// ---- CNC Beckhoff/3 Control/HLI3_GetChannelActiveG.TcPOU
FUNCTION_BLOCK HLI3_GetChannelActiveG
VAR_INPUT
	bExec:	   BOOL;			// riding edge to start read
	nChanIdx: INT;    			// zero based channel index	
END_VAR
VAR_OUTPUT
	ActiveG : ARRAY[0..39] OF INT;
	bBusy: BOOL;
	bError: BOOL;
	nErrorID: UDINT;
END_VAR
VAR
	fbAdsRead: ADSREAD;
END_VAR

(* ========================================================= *)
(*    FUN: HLI3_GetChannelActiveG                   		 *)
(* --------------------------------------------------------- *)
(*   Desc: Gets the channel specific active G functions      *)
(*															 *)
(* Return: Array[0..39] filled with the G information (<> -1)*)
(* Author: MiB                                               *)
(*   Date: 12.01.2016                                        *)
(*   Rev.: 1.0                                               *)
(* ========================================================= *)

fbAdsRead(
	NETID:= '' , 
	PORT:= 553, 
	IDXGRP:= 16#20100 + INT_TO_UDINT(nChanIdx) + 1, 
	IDXOFFS:= 16#3C , 
	LEN:= SIZEOF(ActiveG) , 
	DESTADDR:= ADR(ActiveG),
	READ:= bExec, 
	TMOUT:= , 
	BUSY=> bBusy, 
	ERR=> bError, 
	ERRID=> nErrorId );

END_FUNCTION_BLOCK

// ---- CNC Beckhoff/3 Control/HLI3_GetChannelMessage.TcPOU
FUNCTION_BLOCK HLI3_GetChannelMessage
VAR_INPUT
	/// Number of channel 
	nChanIdx: INT;
	bExecute: BOOL := FALSE;
	bShowDlg: BOOL := FALSE;
END_VAR
VAR_OUTPUT
	strToPLC: STRING(HLI_MSG_CONTENT_STRL) := '';
	iMsgType: DWORD := 0;
END_VAR
VAR
	pChannel: POINTER TO HIGH_LEVEL_INTERFACE_CH;
	pMsgCU: POINTER TO MC_CONTROL_MSG_UNIT;
	pMsgToPLC: POINTER TO STRING(HLI_MSG_CONTENT_STRL);
END_VAR

(* ========================================================= *)
(*     FB: HLI_GetChannelMessage                             *)
(* --------------------------------------------------------- *)
(*   Desc: Get message from the CNC                          *)
(*   Author: MK, MiB                                         *)
(*   Date: 20.11.2012                                        *)
(*   Last:                                                   *)
(*   Rev.: 1.01                                              *)
(* ========================================================= *)

IF NOT HLI3_CheckChannelValid(nChannel := nChanIdx) THEN
	RETURN;
END_IF


(* Get pointer to data of a specific channel at the HLI *)
pChannel := gpCh[nChanIdx];

(* Control unit at the HLI that handles channel specific messages *)
pMsgCU := ADR(pChannel^.msg_mc_control);

IF bExecute = TRUE THEN
	(* Is the complete message in the control unit? *)
	IF pMsgCU^.request_semaphor_rw = TRUE
	THEN
		(* Pointer to content of the message sent to the PLC *)
		pMsgToPLC := ADR(pMsgCU^.request_r.inhalt);

		(* Get the message from the control unit *)
		strToPLC := pMsgToPLC^;

   	    CNCSystem.Channel[nChanIdx].Message := strToPLC;

		(* Get the message type *)
		iMsgType := pMsgCU^.request_r.typ;

		(* Pop up dialog with the message send to the PLC *)
		IF bShowDlg THEN
			ADSLOGSTR( msgCtrlMask := ADSLOG_MSGTYPE_MSGBOX OR ADSLOG_MSGTYPE_LOG,
			           msgFmtStr   := 'Message sent to PLC via HLI:%s',
			           strArg      := strToPLC);
		END_IF

		(* Acknowledge that you got the message *)
		pChannel^.msg_mc_control.request_semaphor_rw  := FALSE;
	END_IF;
END_IF;

END_FUNCTION_BLOCK

// ---- CNC Beckhoff/3 Control/HLI3_GetEtherCATAxisInfo.TcPOU
FUNCTION HLI3_GetEtherCATAxisInfo : ST_DriveRef
VAR
	arrTemp: ARRAY[1..24] OF BYTE;
	arrNetIdAchse2: ARRAY[0..MAX_STRING_LENGTH] OF BYTE;
	i: INT;
	id: DINT;
	nCha: UINT;
	nPort: UINT;
END_VAR
VAR_INPUT
	nHliAxisIdx: INT;
END_VAR

(* ========================================================= *)
(*    FUN: HLI_GetEtherCATAxisInfo                   		 *)
(* --------------------------------------------------------- *)
(*   Desc: Gets the information about a SoE Drive (Ax5000)   *)
(*  benötigt: TcEtherCAT.lib   *)
(* Return: Structure with the information for the drive     *)
(* Author: MiB                                               *)
(*   Date: 20.11.2012                                        *)
(*   Rev.: 1.2                                               *)
(* ========================================================= *)


IF NOT HLI3_CheckAxisValid(nHliAxisIdx := nHliAxisIdx) THEN
	HLI3_GetEtherCATAxisInfo.sNetId := '';
	HLI3_GetEtherCATAxisInfo.nDriveNo := 0;
	HLI3_GetEtherCATAxisInfo.nSlaveAddr := 0;
	RETURN;	
END_IF


HLI3_GetEtherCATAxisInfo.sNetId := gpAx[nHliAxisIdx]^.lr_state.twincat_box.ads_netid_r;
HLI3_GetEtherCATAxisInfo.nDriveNo := UINT_TO_BYTE(gpAx[nHliAxisIdx]^.lr_state.twincat_box.channel_r);
HLI3_GetEtherCATAxisInfo.nSlaveAddr :=gpAx[nHliAxisIdx]^.lr_state.twincat_box.ads_port_r;

RETURN;

END_FUNCTION

// ---- CNC Beckhoff/3 Control/HLI3_GetFeedholdState.TcPOU
FUNCTION HLI3_GetFeedholdState : BOOL
VAR_INPUT
	/// Number of channel 
	nChanIdx: INT;
END_VAR


IF NOT HLI3_CheckChannelValid(nChannel := nChanIdx) THEN
	RETURN;
END_IF
HLI3_GetFeedholdState:=gpCh[nChanIdx]^.bahn_mc_control.feedhold.state_r;

END_FUNCTION

// ---- CNC Beckhoff/3 Control/HLI3_GetIpoState.TcPOU
FUNCTION HLI3_GetIpoState : BOOL
VAR_INPUT
	nChanIdx: INT;
END_VAR



IF NOT HLI3_CheckChannelValid(nChannel := nChanIdx) THEN
	RETURN;
END_IF

HLI3_GetIpoState:=gpCh[nChanIdx]^.bahn_state.interpolation_active_r;

END_FUNCTION

// ---- CNC Beckhoff/3 Control/HLI3_SetAxisGantryOn.TcPOU
FUNCTION HLI3_SetAxisGantryOn : BOOL
VAR_INPUT
	nHliAxisIdx: INT;
	bEnable: BOOL;
END_VAR

(****************************************************************************************)
(* POU:		HLI_SetAxisGantryOn                      									*)
(* Type:	Function																	*)
(* Author: 	HR																			*)
(* Date: 	11/01/24																	*)
(* Rev.: 	1.0																			*)
(* ------------------------------------------------------------------------------------ *)
(* Desc:	Enables the axis specific control unit for driving out the gantry			*)
(*			difference. The actual movement is triggered by the input 'bEnable'.		*)
(*			The current axis has to be a gantry slave. That means:						*)
(*				+ It is not attached to a channel										*)
(*				+ kenngr.achs_mode		0x2000n		(where n specifies the axis type)	*)
(*				+ kenngr.gantry_ax_nr	1			(e. g. axis no. of gantry master)	*)
(*				+ kenngr.gantry_offset  10000		(e. g. difference to be driven out)	*)
(*				+ kenngr.gantry_vb_korr	20000		(e. g. velocity for driving out)	*)
(****************************************************************************************)

(* Check specified logical axis no first *)
IF NOT HLI3_CheckAxisValid(nHliAxisIdx := nHliAxisIdx) THEN
	HLI3_SetAxisGantryOn := FALSE;
	RETURN;
END_IF

gpAx[nHliAxisIdx]^.lr_mc_control.gantry_on.enable_w	:= TRUE;
gpAx[nHliAxisIdx]^.lr_mc_control.gantry_on.command_w	:= bEnable;
HLI3_SetAxisGantryOn	:= TRUE;

END_FUNCTION

// ---- CNC Beckhoff/3 Control/HLI3_SetAxisReferenceCam.TcPOU
FUNCTION HLI3_SetAxisReferenceCam : BOOL
VAR_INPUT
	nHliAxisIdx: INT;
	bReferenceCam: BOOL;
END_VAR
VAR
	/// Index of axis specific HLI area 
	nHliAxIfcIdx: INT;
END_VAR

(* ========================================================= *)
(*    FUN: HLI_SetAxisReferenceCam                           *)
(* --------------------------------------------------------- *)
(*   Desc:                                                   *)
(* Author: MK,MiB                                            *)
(*   Date: 30.11.2012                                        *)
(*   Rev.: 1.1                                               *)
(* ========================================================= *)


IF NOT HLI3_CheckAxisValid(nHliAxisIdx := nHliAxisIdx) THEN
	HLI3_SetAxisReferenceCam := FALSE;
	RETURN;
END_IF

(* set reference cam *)
gpAx[nHliAxisIdx]^.lr_mc_control.reference_cam.enable_w  := TRUE;
gpAx[nHliAxisIdx]^.lr_mc_control.reference_cam.command_w := bReferenceCam;

HLI3_SetAxisReferenceCam := TRUE;

END_FUNCTION

// ---- CNC Beckhoff/3 Control/HLI3_SetAxisReferencePosition.TcPOU
FUNCTION HLI3_SetAxisReferencePosition : BOOL
VAR_INPUT
	bSetRefpos: BOOL;
	nHliAxisIdx: INT;
END_VAR

(* ========================================================= *)
(*    FUN: HLI_SetAxisReferenceposition                      *)
(* --------------------------------------------------------- *)
(*   Desc:                                                   *)
(* Author: HR                                                *)
(*   Date: 09.11.2010                                        *)
(*   Rev.: 1.0                                               *)
(* ========================================================= *)
HLI3_SetAxisReferencePosition := FALSE;

IF NOT HLI3_CheckAxisValid(nHliAxisIdx := nHliAxisIdx) THEN	
	RETURN;
END_IF

(* set reference position *)
gpAx[nHliAxisIdx]^.lr_mc_control.set_reference_position.command_w := bSetRefpos;
HLI3_SetAxisReferencePosition := TRUE;

END_FUNCTION

// ---- CNC Beckhoff/3 Control/HLI3_SetAxisSpindleStopAtProgramEnd.TcPOU
FUNCTION_BLOCK HLI3_SetAxisSpindleStopAtProgramEnd
VAR_INPUT
	bExecute: BOOL;
	bSpindelStopAtProgramEnd: BOOL;
	nHliAxisIdx: INT;
END_VAR
VAR_OUTPUT
	bBusy: BOOL;
END_VAR
VAR
	/// Index of axis specific HLI area 
	nHliAxIfcIdx: INT;
	nState: INT;
	fbRTrigExecute: R_TRIG;
END_VAR

(****************************************************************************************)
(* POU:		HLI_SetAxisSpindleStopAtProgramEnd                      					*)
(* Type:		FB																		*)
(* Author: 	HR                                              							*)
(* Date: 	24.01.11																	*)
(* Rev.: 	1.0                                               							*)
(* ------------------------------------------------------------------------------------ *)
(* Desc:	Check wether the axis specified by input 'nLogAxisNo' is a spindle and 		*)
(*			(re-) sets (depending on the state of input 'bSpindelStopAtProgramEnd') 	*)
(*			the spindle stop feature on the HLI.										*)
(****************************************************************************************)

(****************************************************************************************)
(*								Check logical axis no									*)
(****************************************************************************************)
IF NOT HLI3_CheckAxisValid(nHliAxisIdx := nHliAxisIdx) THEN	
	RETURN;
END_IF
(****************************************************************************************)
(*									Build trigger										*)
(****************************************************************************************)
fbRTrigExecute
	(CLK := bExecute);

(****************************************************************************************)
(*								   (Re-)set sequence									*)
(****************************************************************************************)
CASE nState OF
 (* ----------------------------------------------------------------------------------- *)
 0: (* INIT STATE  *)
  	bBusy			:= FALSE;

	IF fbRTrigExecute.Q THEN
		bBusy		:= TRUE;
		nState		:= 10;
	END_IF

 (* ----------------------------------------------------------------------------------- *)
 10: (* ENABLE THE CONTROL UNIT IF THE AXIS IS A SPINDLE *)

	IF gpAx[nHliAxisIdx]^.ipo_state.spindle_axis_r THEN
		gpAx[nHliAxisIdx]^.ipo_mc_control.spdl_stop_at_prog_end.enable_w := TRUE;
		nState 		:= 20;
	ELSE
		nState 		:= 0;
	END_IF

 (* ---------------------------------------------------------------------------------- *)
 20: (* (RE-) SET SPINDLE STOP FUNCTION *)
	gpAx[nHliAxisIdx]^.ipo_mc_control.spdl_stop_at_prog_end.command_w := bSpindelStopAtProgramEnd;
	nState 			:= 0;
END_CASE

END_FUNCTION_BLOCK

// ---- CNC Beckhoff/3 Control/HLI3_SetAxisTrackingOperation.TcPOU
FUNCTION HLI3_SetAxisTrackingOperation : BOOL
VAR_INPUT
	nHliAxisIdx: INT;
	bPLCAxisEnable: BOOL;
END_VAR

(* ========================================================= *)
(*    FUN: HLI_SetAxisTrackingOperation                      *)
(* --------------------------------------------------------- *)
(*   Desc:                                                   *)
(*   Author: TV                                              *)
(*   Date: 15.09.2006                                        *)
(*   Rev.: 1.0                                               *)
(*         1.1 13.08.2013 Nachführbetrieb nicht bei Achsfehler einschalten *)
(* ========================================================= *)

IF NOT HLI3_CheckAxisValid(nHliAxisIdx := nHliAxisIdx) THEN	
	HLI3_SetAxisTrackingOperation := FALSE;
	RETURN;
END_IF

(* tracking operation (follow up) on / off *)
IF NOT bPLCAxisEnable THEN
	gpAx[nHliAxisIdx]^.lr_mc_control.follow_up.command_w := TRUE;
		HLI3_SetAxisTrackingOperation := TRUE;
ELSE
	gpAx[nHliAxisIdx]^.lr_mc_control.follow_up.command_w := FALSE;
		HLI3_SetAxisTrackingOperation := FALSE;
END_IF

END_FUNCTION

// ---- CNC Beckhoff/3 Control/HLI3_SetProbingSignal.TcPOU
FUNCTION HLI3_SetProbingSignal : BOOL
VAR_INPUT
	nHliAxisIdx: INT;
	bProbingSignal: BOOL;
END_VAR


IF NOT HLI3_CheckAxisValid(nHliAxisIdx := nHliAxisIdx) THEN	
	HLI3_SetProbingSignal := FALSE;
	RETURN;
END_IF


gpAx[nHliAxisIdx]^.lr_mc_control.probing_signal.enable_w  := TRUE;
gpAx[nHliAxisIdx]^.lr_mc_control.probing_signal.command_w := bProbingSignal;
HLI3_SetProbingSignal := TRUE;

END_FUNCTION

// ---- CNC Beckhoff/4 MHT-Function/HLI3_QuitAxisMFunction.TcPOU
FUNCTION HLI3_QuitAxisMFunction : BOOL
VAR_INPUT
	/// Number of axis 
	nHliAxisIdx: INT;
END_VAR
VAR
	/// Data of a M/H techno unit 
	pMHProcess: POINTER TO HLI_M_H_PROZESS;
	/// Data of a spindle unit 
	pSProcess: POINTER TO HLI_S_PROZESS;
	/// Data of a techno unit 
	pTProcess: POINTER TO HLI_T_PROZESS;
	/// local pointer to Data of actual Axis 
	pAxisData: POINTER TO HIGH_LEVEL_INTERFACE_AX;
	/// local pointer to actual techno unit 
	pActTechnoUnit: POINTER TO TECHNO_UNIT_AX;
	/// loop variable 
	idx: UINT;
	/// Index of axis specific technology function at HLI 
	nTechFctMaxIdx: UINT;
	/// basis id of a tool 
	nToolBasicId: UDINT;
	/// spindle movement command 
	SpdlMoveCmd: UINT;
	/// SpindleRevolution 
	Revolution: UDINT;
	/// SpindleRevolution 
	pRevolution: POINTER TO UDINT;
	/// Number of M-function 
	FuncNr: UDINT;
END_VAR

(* ========================================================= *)
(*    FUN: HLI_QuitAxisMFunction                             *)
(* --------------------------------------------------------- *)
(*   Desc:                                                   *)
(* Author: MK                                                *)
(*   Rev.: 1.1                                               *)
(*   Date: 18.07.2002                                        *)
(*       : 08.04.2005                                        *)
(* ========================================================= *)

HLI3_QuitAxisMFunction := FALSE;
IF NOT (HLI3_CheckAxisValid(nHliAxisIdx := nHliAxisIdx)) THEN
	RETURN;
END_IF


(* get pointer to Axis data *)
pAxisData := gpAx[nHliAxisIdx];

(* test if there are open synchronisations  *)
IF pAxisData^.used_units_std_sync_r > 0 THEN

	nTechFctMaxIdx := pAxisData^.used_units_std_sync_r - 1;

	FOR idx := 0 TO nTechFctMaxIdx DO
	
		(* get pointer to actual techno unit *)
		pActTechnoUnit := ADR(pAxisData^.techno_unit_std_sync[idx]);
	
		(* test if this M-function has to be acknowledged *)
		IF pActTechnoUnit^.please_rw = TRUE AND				(* request from CNC *)
			pActTechnoUnit^.done_w = FALSE					(* not acknowledged *)
		THEN
	
			IF pActTechnoUnit^.fkt_ctrl_r = HLI_INTF_M_FKT THEN
				(* Example: read number of M-function *)
				pMHProcess := ADR(pActTechnoUnit^.attribut_r.data[0]);
				FuncNr := pMHProcess^.nr;
				ADSLOG(strMsg:='Axis acknowledge of M-function: %d', nDINT:=UDINT_TO_DINT(FuncNr), strArg:='');
			ELSE
				IF pActTechnoUnit^.fkt_ctrl_r = HLI_INTF_SPINDEL THEN (* spindle-fuction *)
					pSProcess := ADR(pActTechnoUnit^.attribut_r.data[0]);
	
					(* Example: read revolution of S-function *)
					Revolution := DINT_TO_UINT(pSProcess^.rev);
					ADSLOG(strMsg:='Spindle S-function: %d', nDINT:=UDINT_TO_DINT(Revolution), strArg:='');
	
					(* Example: read number of S-function *)
					SpdlMoveCmd := pSProcess^.move_cmd;
					ADSLOG(strMsg:='Spindle acknowledge of M-function: %d', nDINT:=SpdlMoveCmd, strArg:='');
				ELSE
					ADSLOGDINT( msgCtrlMask :=    ADSLOG_MSGTYPE_MSGBOX
					                           OR ADSLOG_MSGTYPE_LOG,
								msgFmtStr   := 'Axis acknowledge unknown type: %d',
								dintArg     := pActTechnoUnit^.fkt_ctrl_r);
				END_IF
			END_IF
	
			(* acknowledge this M-function *)
			pActTechnoUnit^.please_rw := FALSE;
			pActTechnoUnit^.done_w := TRUE;
	
			HLI3_QuitAxisMFunction := TRUE;
		END_IF
	END_FOR

END_IF

END_FUNCTION

// ---- CNC Beckhoff/4 MHT-Function/PRG_FastMFunctions.TcPOU
PROGRAM PRG_FastMFunctions
VAR
	anMFunctionNo						: ARRAY[0..MAX_FAST_M_FUNC_ITEM_IDX] OF UINT;
	
	fbFastMFunctionProvider				: HLI3_FastMFunctionProvider;
	fbFastMFunctionHandler				: HLI3_FastMFunctionHandler;
	
	(* abyOutput					AT %Q*	: ARRAY[0..MAX_FAST_M_FUNC_OUTPUT_IDX] OF BYTE; *) 
	abyOutput					: ARRAY[0..MAX_FAST_M_FUNC_OUTPUT_IDX] OF BYTE; (* Demo output, if needed use the line above *)

END_VAR

(****************************************************************************************)
(* POU:		PRG_FastMFunctions                    										*)
(* Type:	PRG																			*)
(* Author: 	RCH		                                             						*)
(* Date: 	14/10/29																	*)
(* Rev.: 	1.0                                               							*)
(* ------------------------------------------------------------------------------------ *)
(* Desc.:	PLC program to demonstrate usage of MOS_TS M functions using the FB´s		*)
(*			HLI3_FastMFunctionProvider and HLI3_FastMFunctionHandler.					*)
(*			In order to achieve a determenistic output behavior this program has to be 	*)
(*			called by a task running synchronously to the CNC GEO task. Therefore that	*)
(*			task´s priority  has to be adjusted in a way that it gets called by the 	*)
(* 			realtime system	right after the CNC GEO task.								*)
(*																						*)
(*			THIS IMPLEMENTATION REQUIRES A 1MS CNC GEO AND 1MS FAST PLC TASK CYCLE!!!	*)
(* ------------------------------------------------------------------------------------ *)
(* Rev.:	<Enter revision number here>												*)
(* Date:	<Enter revision data here>				                                   	*)
(* Author:	<Enter author´s shortcut here>											 	*)
(* Desc.:	<Enter description here>													*)
(****************************************************************************************)


(****************************************************************************************)
(*	  						Configure M function no´s to provide						*)
(****************************************************************************************)
(* Add up to MAX_FAST_M_FUNC_ITEM_IDX m function numbers that should be handled by 		*)
(* fbFastMFunctionProvider.																*)
anMFunctionNo[0]	:= 25;
anMFunctionNo[1]	:= 26;

fbFastMFunctionProvider
	(nHliChanIdx	:= 0, 
	 anMFunctionNo	:= anMFunctionNo
	);
	
(****************************************************************************************)
(*	  						 	Handle Laser ON/OFF (M25/M26)							*)
(****************************************************************************************)
(* M function numbers for switching ON and OFF have to be contained in the 				*)
(* 'anMFunctionNo' array of the HLI3_FastMFunctionProvider instance which provides the	*)
(* 'stData' structure to this FB.														*)
(* The delay times nDelayOn and nDelayOff can be used to adopt to external hardware		*)
(* delays!																				*)
fbFastMFunctionHandler
	(bForceOff		:= FALSE, 
	 bReset			:= FALSE, 
	 nFunctionNoOn	:= 25, 
	 nDelayOn		:= 0,			
	 nFunctionNoOff	:= 26, 
	 nDelayOff		:= 0,
	 stData			:= fbFastMFunctionProvider.stData,
	 abyOutput		=> abyOutput
	);

END_PROGRAM

// ---- CNC Beckhoff/5 Variables/HLI3_GetVEChannelDIntValue.TcPOU
FUNCTION HLI3_GetVEChannelDIntValue : DINT
VAR_INPUT
	/// HLI Channel Index 
	nChanIdx: INT;
	/// Index of variable  range 1 ...     HLI_VE_VALUEMAX 
	nVEIndex: DINT;
	/// Array index. 0 if no array 
	nArrayIndex: DINT := 0;
	/// serves acess to the global variable array 
	bGlobal: BOOL;
END_VAR
VAR
	pVeData: POINTER TO VEData := 0;
	/// Size of the datatype of the returned value 
	iDatatypeSize: DINT;
	ptr: POINTER TO DINT;
	ChIdx: UDINT;
	SizeField: DINT := 0;
END_VAR

(* ========================================================= *)
(*    FUN: GetVEChannelDINTValue                            *)
(* --------------------------------------------------------- *)
(*   Desc: Reads a V.E.Variable of DINT                    *)
(* 	 Author: CL  / TV                                        *)
(*   Date: 16.05.2006                                        *)
(*   Last: 28.01.2013                                        *)
(*   Rev.: 1.3                                               *)
(* ========================================================= *)

IF  nVEIndex >= 0 AND
	nArrayIndex >= 0 THEN

	(* test if channel specific or global *)
	IF bGlobal = FALSE  THEN
		IF NOT HLI3_CheckChannelValid(nChannel := nChanIdx) THEN
			RETURN;
		END_IF
				
		pVeData := gpVECh[nChanIdx];
	ELSE
		pVeData := gpVEGlobal;
	END_IF

	IF pVeData <> 0 THEN
		IF pVeData <> 0 THEN
			iDatatypeSize := SIZEOF(ptr^);
                         	ptr := pVeData +  24  * nVEIndex + (iDatatypeSize * nArrayIndex);
                           HLI3_GetVEChannelDIntValue := ptr^; (* successfully completed return *)
                END_IF
	END_IF
END_IF

END_FUNCTION

// ---- CNC Beckhoff/5 Variables/HLI3_GetVEChannelBooleanValue.TcPOU
FUNCTION HLI3_GetVEChannelBooleanValue : BOOL
VAR_INPUT
	/// HLI Channel Index
	nChanIdx: INT;
	/// Index of variable  range 1 ...     HLI_VE_VALUEMAX 
	nVEIndex: DINT;
	/// Array index. 0 if no array 
	nArrayIndex: DINT := 0;
	/// serves acess to the global variable array 
	bGlobal: BOOL;
END_VAR
VAR
	pVeData: POINTER TO VEData := 0;
	/// Size of the datatype of the returned value 
	iDatatypeSize: DINT;
	ptr: POINTER TO BOOL;
	ChIdx: UDINT;
	SizeField: DINT := 0;
END_VAR

(* ========================================================= *)
(*    FUN: GetVEChannelDINTValue                            *)
(* --------------------------------------------------------- *)
(*   Desc: Reads a V.E.Variable of Boolean                   *)
(* 	 Author: CL  / TV                                        *)
(*   Date: 16.05.2006                                        *)
(*   Last: 05.12.2013                                        *)
(*   Rev.: 1.3                                               *)
(* ========================================================= *)

IF  nVEIndex >= 0 AND
	nArrayIndex >= 0 THEN

	(* test if channel specific or global *)
	IF bGlobal = FALSE  THEN
		IF NOT HLI3_CheckChannelValid(nChannel := nChanIdx) THEN
			RETURN;
		END_IF
				
		pVeData := gpVECh[nChanIdx];
	ELSE
		pVeData := gpVEGlobal;
	END_IF

	IF pVeData <> 0 THEN
		IF pVeData <> 0 THEN
			iDatatypeSize := SIZEOF(ptr^);
                         	ptr := pVeData +  24  * nVEIndex + (iDatatypeSize * nArrayIndex);
                           HLI3_GetVEChannelBooleanValue := ptr^; (* successfully completed return *)
                END_IF
	END_IF
END_IF

END_FUNCTION

// ---- CNC Beckhoff/5 Variables/HLI3_GetVEChannelLRealValue.TcPOU
FUNCTION HLI3_GetVEChannelLRealValue : LREAL
VAR_INPUT
	/// HLI Channel Index
	nChanIdx: INT;
	/// Index of variable  range 1 ...     HLI_VE_VALUEMAX 
	nVEIndex: DINT;
	/// Array index. 0 if no array 
	nArrayIndex: DINT := 0;
	/// serves acess to the global variable array 
	bGlobal: BOOL;
END_VAR
VAR
	pVeData: POINTER TO VEData := 0;
	/// Size of the datatype of the returned value 
	iDatatypeSize: DINT;
	ptr: POINTER TO LREAL;
	ChIdx: UDINT;
	SizeField: DINT := 0;
END_VAR

(* ========================================================= *)
(*    FUN: GetVEChannelLrealValue                            *)
(* --------------------------------------------------------- *)
(*   Desc: Reads a V.E.Variable of REAL64                    *)
(* 	 Author: CL  / TV                                        *)
(*   Date: 16.05.2006                                        *)
(*   Last: 28.01.2013                                        *)
(*   Rev.: 1.3                                               *)
(* ========================================================= *)

IF  nVEIndex >= 0 AND
	nArrayIndex >= 0 THEN

	(* test if channel specific or global *)
	IF bGlobal = FALSE  THEN
		IF NOT HLI3_CheckChannelValid(nChannel := nChanIdx) THEN
			RETURN;
		END_IF
				
		pVeData := gpVECh[nChanIdx];
	ELSE
		pVeData := gpVEGlobal;
	END_IF

	IF pVeData <> 0 THEN
		IF pVeData <> 0 THEN
			iDatatypeSize := SIZEOF(ptr^);
                         	ptr := pVeData +  24  * nVEIndex + (iDatatypeSize * nArrayIndex);
                           HLI3_GetVEChannelLRealValue := ptr^; (* successfully completed return *)
                END_IF
	END_IF
END_IF

END_FUNCTION

// ---- CNC Beckhoff/5 Variables/HLI3_GetVEChannelStringValue.TcPOU
FUNCTION HLI3_GetVEChannelStringValue : STRING(23)
VAR_INPUT
	/// HLI Channel Index
	nChanIdx: INT;
	/// Index of variable  range 1 ...     HLI_VE_VALUEMAX 
	nVEIndex: DINT;
	/// Array index. 0 if no array 
	nArrayIndex: DINT := 0;
	/// serves acess to the global variable array 
	bGlobal: BOOL;
END_VAR
VAR
	pVeData: POINTER TO VEData := 0;
	/// Size of the datatype of the returned value 
	iDatatypeSize: DINT;
	ptr: POINTER TO STRING(24);
	ChIdx: INT;
END_VAR

(* ========================================================= *)
(*    FUN: GetVEChannelStringValue                           *)
(* --------------------------------------------------------- *)
(*   Desc: Reads a V.E.Variable of STRING                    *)
(* 	 Author: CL / TV                                         *)
(*   Date: 16.05.2006                                        *)
(*   Last: 28.01.013                                        *)
(*   Rev.: 1.1                                               *)
(* ========================================================= *)

(* Config Example
	VAR[0].name                                           StringValue
	VAR[0].index                                           1
	VAR[0].TYPE                                           STRING
	VAR[0].scope                                          GLOBAL
	VAR[0].synchronisation                                TRUE
	VAR[0].access_rights                                  READ_WRITE
	VAR[0].array_size                                     21
	VAR[0].size                                           24
	VAR[0].create_hmi_interface                           0
*)

IF  nVEIndex >= 0 AND
	nArrayIndex >= 0 THEN

	(* test if channel specific or global *)
	IF bGlobal = FALSE  THEN
		IF NOT HLI3_CheckChannelValid(nChannel := nChanIdx) THEN
			RETURN;
		END_IF
		pVeData := gpVECh[nChanIdx];
	ELSE
		pVeData := gpVEGlobal;
	END_IF

	IF pVeData <> 0 THEN
		 IF pVeData <> 0 THEN
			iDatatypeSize := SIZEOF(ptr^);
			iDatatypeSize := 24;
            ptr := pVeData +  24  * nVEIndex + (iDatatypeSize * nArrayIndex);
            HLI3_GetVEChannelStringValue := ptr^; (* successfully completed return *)
         END_IF
	END_IF
END_IF

END_FUNCTION

// ---- CNC Beckhoff/5 Variables/HLI3_LinkVEChannelStructure.TcPOU
FUNCTION HLI3_LinkVEChannelStructure : POINTER TO DWORD
VAR_INPUT
	/// HLI Channel Index 
	nChanIdx: INT;	
	/// serves acess to the global variable array 
	bGlobal: BOOL;
END_VAR
VAR
	pVeData: POINTER TO VEData := 0;
	ptr: POINTER TO DWORD;
	ChIdx: UDINT;
	nVEIndex: POINTER TO DWORD;
END_VAR

(* ========================================================= *)
(*    FUN: LinkVEChannelStructure                            *)
(* --------------------------------------------------------- *)
(*   Desc: Link VE variable to the memory of the CNC         *)
(*   Author: CL, MK                                            *)
(*   Date: 16.05.2006                                        *)
(*   Rev.: 1.3                                               *)
(*       : MK  access changed                                *)
(*		   1.2												 *)
(*		   MiB 7.11.2012 check zero pointers				 *)
(*		   TV 19.08.2015 Input Parm. nIndex removed          *) 
(* ========================================================= *)

	(* test if channel specific or global *)
     IF bGlobal THEN
    	IF gpVEGlobal = 0  THEN   (* check for  zero pointer *)
        	RETURN; (* Cancel *)
        END_IF
			pVeData := gpVEGlobal;
	 ELSE
		IF NOT HLI3_CheckChannelValid(nChannel := nChanIdx) THEN
			RETURN;
		END_IF
							
		pVeData := gpVECh[nChanIdx];
	END_IF 

	IF pVeData <> 0 THEN
    	ptr := pVeData;
		HLI3_LinkVEChannelStructure := ptr; (* successfully completed return *)
	END_IF

END_FUNCTION

// ---- CNC Beckhoff/5 Variables/HLI3_SetVEChannelDIntValue.TcPOU
FUNCTION HLI3_SetVEChannelDIntValue : BOOL
VAR_INPUT
	/// HLI Channel Index
	nChanIdx: INT;
	/// Index of variable  range 1 ...     HLI_VE_VALUEMAX 
	nVEIndex: DINT;
	/// Array index. 0 if no array 
	nArrayIndex: DINT := 0;
	/// serves acess to the global variable array 
	bGlobal: BOOL;
	/// Value to be written 
	val: DINT;
END_VAR
VAR
	pVeData: POINTER TO VEData := 0;
	/// Size of the datatype of the returned value 
	iDatatypeSize: DINT;
	ptr: POINTER TO DINT;
	ChIdx: UDINT;
	SizeField: DINT := 0;
END_VAR

(* ========================================================= *)
(*    FUN: SetVEChannelDIntValue                           *)
(* --------------------------------------------------------- *)
(*   Desc: Writes a V.E.Variable of REAL64                    *)
(* 	 Author: CL  / TV                                        *)
(*   Date: 16.05.2006                                        *)
(*   Last: 28.01.2013                                        *)
(*   Rev.: 1.3                                               *)
(* ========================================================= *)

IF  nVEIndex >= 0 AND
	nArrayIndex >= 0 THEN

	(* test if channel specific or global *)
	IF bGlobal = FALSE  THEN
		IF NOT HLI3_CheckChannelValid(nChannel := nChanIdx) THEN
			RETURN;
		END_IF
				
		pVeData := gpVECh[nChanIdx];
	ELSE
		pVeData := gpVEGlobal;
	END_IF

	IF pVeData <> 0 THEN
		IF pVeData <> 0 THEN
			iDatatypeSize := SIZEOF(ptr^);
            ptr := pVeData +  24  * nVEIndex + (iDatatypeSize * nArrayIndex);
			ptr^:=val;
            HLI3_SetVEChannelDIntValue := TRUE; (* successfully completed return *)						  						   
       	END_IF
	END_IF
END_IF

END_FUNCTION

// ---- CNC Beckhoff/5 Variables/HLI3_SetVEChannelBooleanValue.TcPOU
FUNCTION HLI3_SetVEChannelBooleanValue : BOOL
VAR_INPUT
	/// HLI Channel Index
	nChanIdx: INT;
	/// Index of variable  range 1 ...     HLI_VE_VALUEMAX 
	nVEIndex: DINT;
	/// Array index. 0 if no array 
	nArrayIndex: DINT := 0;
	/// serves acess to the global variable array 
	bGlobal: BOOL;
	/// Value to be written 
	val: BOOL;
END_VAR
VAR
	pVeData: POINTER TO VEData := 0;
	/// Size of the datatype of the returned value 
	iDatatypeSize: DINT;
	ptr: POINTER TO BOOL;
	ChIdx: UDINT;
	SizeField: DINT := 0;
END_VAR

(* ========================================================= *)
(*    FUN: SetVEChannelDIntValue                           *)
(* --------------------------------------------------------- *)
(*   Desc: Writes a V.E.Variable of REAL64                    *)
(* 	 Author: CL  / TV                                        *)
(*   Date: 16.05.2006                                        *)
(*   Last: 05.12.2013                                        *)
(*   Rev.: 1.3                                               *)
(* ========================================================= *)

IF  nVEIndex >= 0 AND
	nArrayIndex >= 0 THEN

	(* test if channel specific or global *)
	IF bGlobal = FALSE  THEN
		IF NOT HLI3_CheckChannelValid(nChannel := nChanIdx) THEN
			RETURN;
		END_IF
				
		pVeData := gpVECh[nChanIdx];
	ELSE
		pVeData := gpVEGlobal;
	END_IF

	IF pVeData <> 0 THEN
		IF pVeData <> 0 THEN
			iDatatypeSize := SIZEOF(ptr^);
            ptr := pVeData +  24  * nVEIndex + (iDatatypeSize * nArrayIndex);
			ptr^:=val;
            HLI3_SetVEChannelBOOLeanValue := TRUE; (* successfully completed return *)						  						   
       	END_IF
	END_IF
END_IF

END_FUNCTION

// ---- CNC Beckhoff/5 Variables/HLI3_SetVEChannelLRealValue.TcPOU
FUNCTION HLI3_SetVEChannelLRealValue : BOOL
VAR_INPUT
	/// HLI Channel Index
	nChanIdx: INT;
	/// Index of variable  range 1 ...     HLI_VE_VALUEMAX 
	nVEIndex: DINT;
	/// Array index. 0 if no array 
	nArrayIndex: DINT := 0;
	/// serves acess to the global variable array 
	bGlobal: BOOL;
	/// Value to be written 
	val: LREAL;
END_VAR
VAR
	pVeData: POINTER TO VEData := 0;
	/// Size of the datatype of the returned value 
	iDatatypeSize: DINT;
	ptr: POINTER TO LREAL;
	ChIdx: UDINT;
	SizeField: DINT := 0;
END_VAR

(* ========================================================= *)
(*    FUN: SetVEChannelLrealValue                           *)
(* --------------------------------------------------------- *)
(*   Desc: Writes a V.E.Variable of REAL64                    *)
(* 	 Author: CL  / TV                                        *)
(*   Date: 16.05.2006                                        *)
(*   Last: 06.03.2012                                        *)
(*   Rev.: 1.3                                               *)
(* ========================================================= *)

IF  nVEIndex >= 0 AND
	nArrayIndex >= 0 THEN

	(* test if channel specific or global *)
	IF bGlobal = FALSE  THEN
		IF NOT HLI3_CheckChannelValid(nChannel := nChanIdx) THEN
			RETURN;
		END_IF
				
		pVeData := gpVECh[nChanIdx];
	ELSE
		pVeData := gpVEGlobal;
	END_IF

	IF pVeData <> 0 THEN
		IF pVeData <> 0 THEN
			iDatatypeSize := SIZEOF(ptr^);
            ptr := pVeData +  24  * nVEIndex + (iDatatypeSize * nArrayIndex);
			ptr^:=val;
            HLI3_SetVEChannelLRealValue := TRUE; (* successfully completed return *)						  						   
       	END_IF
	END_IF
END_IF

END_FUNCTION

// ---- CNC Beckhoff/5 Variables/HLI3_SetVEChannelStringValue.TcPOU
FUNCTION HLI3_SetVEChannelStringValue : BOOL
VAR_INPUT
	/// HLI Channel Index
	nChanIdx: INT;
	/// Index of variable  range 1 ...     HLI_VE_VALUEMAX 
	nVEIndex: DINT;
	/// Array index. 0 if no array 
	nArrayIndex: DINT := 0;
	/// Value to be written 
	val: STRING(23);
	/// serves acess to the global variable array 
	bGlobal: BOOL;
END_VAR
VAR
	pVeData: POINTER TO VEData := 0;
	/// Size of the datatype of the returned value 
	iDatatypeSize: DINT;
	ptr: POINTER TO STRING;
	ChIdx: INT;
END_VAR

(* ========================================================= *)
(*    FUN: SetVEChannelStringValue                           *)
(* --------------------------------------------------------- *)
(*   Desc: Writes a V.E.Variable of STRING                   *)
(* 	 Author: CL / TV                                         *)
(*   Date: 16.05.2006                                        *)
(*   Last : 13.12.2012										 *)
(*   Rev.: 1.1                                               *)
(* ========================================================= *)

(* Config Example
	VAR[0].name                                           StringValue
	VAR[0].index                                           1
	VAR[0].TYPE                                           STRING
	VAR[0].scope                                          GLOBAL
	VAR[0].synchronisation                                TRUE
	VAR[0].access_rights                                  READ_WRITE
	VAR[0].array_size                                     21
	VAR[0].size                                           24
	VAR[0].create_hmi_interface                           0
*)

IF  nVEIndex >= 0 AND
	nArrayIndex >= 0 THEN

	(* test if channel specific or global *)
	IF bGlobal = FALSE  THEN
		IF NOT HLI3_CheckChannelValid(nChannel := nChanIdx) THEN
			RETURN;
		END_IF
				
		pVeData := gpVECh[nChanIdx];
	ELSE
		pVeData := gpVEGlobal;
	END_IF

	IF pVeData <> 0 THEN
		iDatatypeSize := SIZEOF(ptr^);
		iDatatypeSize := 24;
        ptr := ADR(pVeData^)  +  24  * nVEIndex + (iDatatypeSize * (nArrayIndex));
        ptr^ := val; (* successfully completed return *)
		HLI3_SetVEChannelStringValue := TRUE;
	END_IF
END_IF

END_FUNCTION

// ---- CNC Beckhoff/9 Mis/FB_WriteCNCZeroOffset.TcPOU
/// ------------------------------------------------------------------------------------ 
/// Desc:	Description																	
///**************************************************************************************
///**************************************************************************************
///	 Write NPV Value directly to CNC core using V.G. Variables via ADS	
///**************************************************************************************
FUNCTION_BLOCK FB_WriteCNCZeroOffset
VAR_INPUT
	/// rising edge to start 
	bExecute: BOOL;
	/// which table, G54=1, G55=2, G55=3, .... 
	nG159Index: BYTE;
	/// Channel Indedx
	nChanIdx: UDINT;
	/// Axis name in channel 
	sAxisName: STRING(95);
	/// value to set 
	lrValue: LREAL;
END_VAR
VAR_OUTPUT
	bBusy: BOOL;
	bError: BOOL;
	nErrorID: UDINT;
END_VAR
VAR
	fbAdsWrite: ADSWRITE;
	stCNCG159VG: ST_CNCG159VG;
END_VAR

stCNCG159VG.dValue := LREAL_TO_DINT(lrValue * 10000);
stCNCG159VG.sTarget := 'V.G.NP[';
stCNCG159VG.sTarget := CONCAT(stCNCG159VG.sTarget, BYTE_TO_STRING(nG159Index));
stCNCG159VG.sTarget := CONCAT(stCNCG159VG.sTarget, '].V.');
stCNCG159VG.sTarget := CONCAT(stCNCG159VG.sTarget,sAxisName);

fbAdsWrite(
	PORT:= 552 ,
	IDXGRP:= 16#22300 + nChanIdx+1,
	IDXOFFS:=16#3F,
	LEN:= SIZEOF(stCNCG159VG) ,
	SRCADDR:=ADR(stCNCG159VG) ,
	WRITE:= bExecute,
	TMOUT:= ,
	BUSY=> bBusy,
	ERR=> bError ,
	ERRID=> nErrorID);

END_FUNCTION_BLOCK

// ---- CNC Beckhoff/9 Mis/FB_WriteCNCZeroOffsetDefault.TcPOU
/// ------------------------------------------------------------------------------------ 
/// Desc:	Description																	
///**************************************************************************************
///**************************************************************************************
///	 Write NPV Default (the active table afetr reset) directly to CNC core using V.G. Variables via ADS	
///**************************************************************************************
FUNCTION_BLOCK FB_WriteCNCZeroOffsetDefault
VAR_INPUT
	/// rising edge to start 
	bExecute: BOOL;
	/// which table, G54=1, G55=2, G55=3, .... 
	nG159Index: BYTE;
	/// Channel Indedx
	nChanIdx: UDINT;
END_VAR
VAR_OUTPUT
	bBusy: BOOL;
	bError: BOOL;
	nErrorID: UDINT;
END_VAR
VAR
	fbAdsWrite: ADSWRITE;
	stCNCG159VG: ST_CNCG159VG;
END_VAR

stCNCG159VG.dValue := nG159Index;
stCNCG159VG.sTarget := 'V.G.NP_DEFAULT';

fbAdsWrite(
	PORT:= 552 ,
	IDXGRP:= 16#22300 + nChanIdx+1,
	IDXOFFS:=16#3F,
	LEN:= SIZEOF(stCNCG159VG) ,
	SRCADDR:=ADR(stCNCG159VG) ,
	WRITE:= bExecute,
	TMOUT:= ,
	BUSY=> bBusy,
	ERR=> bError ,
	ERRID=> nErrorID);

END_FUNCTION_BLOCK

// ---- CNC Beckhoff/9 Mis/HLI3_CheckCNCAlive.TcPOU
PROGRAM HLI3_CheckCNCAlive
VAR_INPUT
	nChanIdx: INT;
END_VAR

VAR
	bMessageDisplayed : BOOL;
END_VAR

(* The assumption is made that the cycle time of the PLC is at least twice as big as the CNC cycle time.

The Cycle time of CNC is displayed in element:
	pMC[1]^.addr^.HLIHeadChannel_Data.LCWatchDogUnit_lc.D_cycle_time_r

remark: Take care if PLC cycle is smaller not to check CNC faster as possible !!!

To simulate failure of CNC set cycle time of PLC smaller than CNC (Resource/task configuration).
*)

// HLI3_CheckCNCAlive := FALSE;
IF NOT HLI3_CheckChannelValid(nChannel := nChanIdx) THEN
	RETURN;
END_IF
 
(* Copy current state of live sign to watchdog state    *)
gpCh[nChanIdx]^.head.lc_watchdog.alive_rw
	:= gpCh[nChanIdx]^.head.lc_watchdog.alive_rw;

IF gpCh[nChanIdx]^.head.lc_watchdog.alive_rw = FALSE AND NOT bMessageDisplayed THEN
	(* PLC detects CNC not alive -> start individual emergency stop within PLC *)
	ADSLOGSTR( msgCtrlMask := ADSLOG_MSGTYPE_ERROR OR
							ADSLOG_MSGTYPE_MSGBOX OR
							ADSLOG_MSGTYPE_LOG,
			msgFmtStr := 'PLC detects CNC not alive: %s',
			strArg := 'channel 1');
			
			bMessageDisplayed := TRUE;
END_IF


(* assign return value *)
//HLI3_CheckCNCAlive := gpCh[nChanIdx]^.head.lc_watchdog.alive_rw;

(* reset live sign for next cycle *)
gpCh[nChanIdx]^.head.lc_watchdog.alive_rw := FALSE;

END_PROGRAM

// ---- CNC Beckhoff/9 Mis/HLI3_GetLogAxisId.TcPOU
FUNCTION HLI3_GetLogAxisId : INT
VAR_INPUT
	nHliAxisIdx: INT;
END_VAR
VAR
	i: INT;
END_VAR

(* ========================================================= *)
(*    FUN: HLI3_GetLogAxisId                            	 *)
(* --------------------------------------------------------- *)
(*   Desc: returns the Log. Axis Idx for a given HLI Index   *)
(*   Author: TV                                              *)
(*   Date: 22.01.2014                                        *)
(*   Rev.: 1.0                                               *)
(* ========================================================= *)
HLI3_GetLogAxisId := -1;
IF NOT HLI3_CheckAxisValid(nHliAxisIdx := nHliAxisIdx) THEN
	RETURN;
END_IF

HLI3_GetLogAxisId := UINT_TO_INT(gpAx[nHliAxisIdx]^.head.log_ax_nr_r);

END_FUNCTION

// ---- CNC Beckhoff/9 Mis/HLI_HandleMessages.TcPOU
FUNCTION_BLOCK HLI_HandleMessages
VAR_INPUT
	/// Enable 
	bEnable: BOOL;
	/// Number of channel 
	nChanIdx: INT;
	/// Channelstruct 
	pChannel: POINTER TO ST_CncChannel;
END_VAR
VAR_OUTPUT
	bNewMessage: BOOL;
	bError: BOOL;
	sMessage: STRING(255);
END_VAR
VAR
	/// Index of channel specific HLI area 

	bFirstCycle: BOOL := TRUE;
	bModeChanged: BOOL;
	nState: USINT;
	nActMode: UDINT;
	dwCncState: DWORD;
	fbRtrigStateStart: R_TRIG;
	pString: POINTER TO STRING(HLI_MSG_CONTENT_STRL);
	fbLog: ADSLOGEVENT;
	stMessageData: TcEvent;
END_VAR
VAR CONSTANT
	sFormat: STRING(2) := '%s';
END_VAR

(******************************************************************************)
(* Name:		HLI_HandleMessages											 	*)
(* Date:		08/12/01													 	*)
(* Author:	H. Rausch (Beckhoff Automation GmbH)							 	*)
(* Ver:		1.0																	*)
(* Desc:		Function block for recieving messages from CNC and passing them to*)
(*				the TwinCAT EventLogger. Only the latest message from CNC is 	*)
(*				active there. The event will be resetted if a new message from	*)
(*				CNC is recieved, the CNC state changes to 'ACTIVE', the CNC mode*)
(*				is changed or the channel is resetted							*)
(*																				*)
(*				Messages are passed as a fill string to the event logger with 	*)
(*				source id 9000 and event id 1. This requires a correspondant 	*)
(*				configuration in the tceventsourcelocation.xml and in an		*)
(*				associated message file!										*)
(* ---------------------------------------------------------------------------*)
(* Rev:		Add new version number here!										*)
(* Date.		Add revision data here											*)
(* Desc:		Add revision description here!									*)
(******************************************************************************)

(* Write event config data once on start up *)
IF bFirstCycle THEN
	stMessageData.bQuitRequired			:= TRUE;
	stMessageData.Class					:= TCEVENTCLASS_MESSAGE;
	stMessageData.DataFormatStrAddress	:= ADR(sFormat);
	stMessageData.Prio					:= 0;
	stMessageData.Id					:= 1;
	stMessageData.SourceId 				:= 9000;
	stMessageData.Flags 				:= TCEVENTFLAG_LOG OR TCEVENTFLAG_SRCID;
	stMessageData.StreamType			:= TCEVENTSTREAM_SIMPLE;
	stMessageData.ProgId 				:= 'TcEventFormatter.TcXmlFormatter';
END_IF



(* Check for zero pointer and leave fb if necessary *)
IF NOT HLI3_CheckChannelValid(nChannel := nChanIdx) THEN
	RETURN;
END_IF
	(* Check CNC state *)
	dwCncState := HLI3_GetChannelState(nChanIdx:=nChanIdx);

	(* Rising trig if CNC state changes to ACTIVE *)
	fbRtrigStateStart
		(CLK := (dwCncState = HLI_IMCM_PROCESS_ACTIVE));

	(* Watch CNC mode *)
	bModeChanged	:= (nActMode <> pChannel^.ActMode);
	nActMode 		:= pChannel^.ActMode;

IF NOT bEnable THEN
	gpCh[nChanIdx]^.msg_mc_control.enable_w				:= FALSE;
	gpCh[nChanIdx]^.msg_mc_control.request_semaphor_rw	:= FALSE;
	sMessage										:= '';
ELSE
	gpCh[nChanIdx]^.msg_mc_control.enable_w 			:= TRUE;

	CASE nState OF
	 0:
		(* Wait for new messages from CNC *)
		IF gpCh[nChanIdx]^.msg_mc_control.request_semaphor_rw THEN
			(* Convert byte stream to string *)
			pString  := ADR(gpCh[nChanIdx]^.msg_mc_control.request_r.inhalt);
			sMessage := pString^;
			(* Reset notification from HLI *)
			gpCh[nChanIdx]^.msg_mc_control.request_semaphor_rw := FALSE;

			nState := 1;
		END_IF

	 1:
		(* Wait that ADSEVENTLOG instance is cleared *)
		IF (fbLog.EventState = 0) THEN
			nState := 2;
		END_IF

	 2:
		(* Set message to eventlogger *)
		IF (fbLog.EventState > 0) THEN
			nState := 0;
		END_IF

	END_CASE

	(* Managing Eventlogger *)
	fbLog
		(NETID				:= '',
		 PORT					:= 110,
		 Event				:= (nState = 2),
		 EventQuit			:= (nState = 1) OR
									(dwCncState = HLI_IMCM_PROCESS_RESETTING) OR
									fbRtrigStateStart.Q OR
									bModeChanged,
		 EventConfigData	:= stMessageData,
		 EventDataAddress	:= ADR(sMessage),
		 EventDataLength	:= SIZEOF(sMessage),
		 TMOUT				:= t#2s
		);
END_IF

(* Reset first cycle indicator *)
bFirstCycle := FALSE;

END_FUNCTION_BLOCK

// ---- CNC Beckhoff/9 Mis/HLI_MoveSpindle.TcPOU
///*********************************************************************************************************
///NAME.......................:	HLI_MoveSpindle	
///DATUM....................:	7.9.2009
///AUTOR....................:	Michael Balsfulland (MiB)
///VERSION................:	1.0
///				1.1 20.8.2010 MiB: kompletter Umbau auf Schrittkette mit Fehlerhandling
///BESCHREIBUNG.:	 Spindel mit einer vorgegeben Geschwindigkeit starten oder Spindel stoppen
///......................: 	
///
///**********************************************************************************************************
FUNCTION_BLOCK HLI_MoveSpindle
VAR
	pUnit: POINTER TO MC_CONTROL_EXT_TO_IPO;
	fbRTrigStart: R_TRIG;
	fbRTrigStop: R_TRIG;
	nState: INT;
	/// Index of axis specific HLI area 
	nHliAxIfcIdx: UDINT;
END_VAR
VAR_INPUT
	/// Spindel Achssnummer 
	nLogAxisNr: UDINT;
	/// U/min 
	nSpeed: DINT;
	/// steigende Flanke 
	bStart: BOOL;
	/// steigende Flanke 
	bStop: BOOL;
END_VAR
VAR_OUTPUT
	bBusy: BOOL;
	bError: BOOL;
	nErrID: INT;
	sErrText: STRING;
END_VAR

fbRTrigStart(clk := bStart);
IF fbRTrigStart.Q THEN
	bError := FALSE;
	nErrId := 0;
	sErrText := '';
	nState := 100;   (* Spindel starten *)
END_IF


fbRTrigStop(clk := bStop);
IF fbRTrigStop.Q THEN
	bError := FALSE;
	nErrId := 0;
	sErrText := '';
	nState := 200;  (* Spindel stoppen *)
END_IF

nHliAxIfcIdx := nLogAxisNr - 1;

IF fbRTrigStop.Q OR fbRTrigStart.Q THEN   (* Grundzustände testen *)
	bBusy := TRUE;
	IF nLogAxisNr = 0 THEN
		nState := -1;
		nErrID := 1;
		sErrText := 'Spindel ID = 0';
	END_IF
	IF ADR(gpAx[nHliAxIfcIdx]^)  = 0  THEN
		nState := -1;
		nErrID := 2;
		sErrText := 'Achsstruktur nicht vorhanden -> eventuell HLI Init nicht OK';
	END_IF
	IF gpAx[nHliAxIfcIdx]^.ipo_state.spindle_axis_r <> TRUE THEN
		nState := -1;
		nErrID := 3;
		sErrText := 'Achse ist kene Spindel';
	END_IF
END_IF

CASE nState OF


-1: (* Fehler *)
   	bError := TRUE;
	bBusy := FALSE;

0: (* IDLE *)
	bBusy := FALSE;


100: (* Spindel starten *)
	(* Check Override *)
	gpAx[nHliAxIfcIdx]^.ipo_mc_control.override.enable_w := TRUE;
	IF gpAx[nHliAxIfcIdx]^.ipo_mc_control.override.state_r = 0 THEN
		nState := -1;
		nErrID := 4;
		sErrText := 'Spindeloverride = 0';
	ELSE
		nState := 110;
	END_IF


110: (* Parametrieren des Aufrufs *)
	pUnit := ADR(gpAx[nHliAxIfcIdx]^.ipo_mc_control.ext_to_ipo);
	IF (nSpeed > 0) THEN
		pUnit^.command_w.vb_prog   :=  nSpeed * 360 / 60 * 1000  ;(*Programmierter Satzvorschub in u/min*)
		pUnit^.command_w.dreh_info := 1;(* rechtslauf *)
	ELSE
		pUnit^.command_w.vb_prog   :=  nSpeed * 360 / 60 * 1000  ;(*Programmierter Satzvorschub in u/min*)
		pUnit^.command_w.dreh_info := 0;(* linkslauf*)
	END_IF
	pUnit^.command_w.geo_gm_fkt    := 0;(*G- und M- Fkt.-Bitleiste*)
	pUnit^.command_w.satz_typ      := HLI_NC_MOVE_ENDLOS;(*Einer der Werte: HLI_NC_MOVE_LIN, HLI_NC_MOVREF, HLI_NC_MOVE_ENDLOS, HLI_NC_SPINDEL_STOP*)
	IF pUnit^.command_semaphor_rw = FALSE THEN
	    pUnit^.command_semaphor_rw := TRUE;
	    nState := 120;
	END_IF

	IF (nSpeed=0) THEN
		nState := -1;
		nErrID := 6;
		sErrText := 'Vorgabegeschwindigkeit = 0';
	END_IF

120: (* Start *)

	IF pUnit^.command_semaphor_rw = FALSE THEN
	    nState := 300;  (* checken Auftragsfehler *)
	END_IF



200: (* Spindel Stopp*)
	pUnit := ADR(gpAx[nHliAxIfcIdx]^.ipo_mc_control.ext_to_ipo);
	pUnit^.command_w.satz_typ  := HLI_NC_SPINDEL_STOP;(*Einer der Werte: HLI_NC_MOVE_LIN, HLI_NC_MOVREF, HLI_NC_MOVE_ENDLOS, HLI_NC_SPINDEL_STOP*)
	pUnit^.command_w.dreh_info := 0;(*Drehinformation*)
	IF pUnit^.command_semaphor_rw = FALSE THEN
	    pUnit^.command_semaphor_rw := TRUE;
	    nState := 210;
	END_IF

210: (* Warten auf Stop *)
	IF pUnit^.command_semaphor_rw = FALSE THEN
	    nState := 300;   (* checken Auftragsfehler *)
	END_IF

300: (* checken Auftragsfehler *)
	IF (gpAx[nHliAxIfcIdx]^.ipo_state.spindle_order_error_r) THEN
		nState := -1;
		nErrID := 5;
		sErrText := 'Beauftragunsfehler Spindel';
	ELSE
		nState := 310;
	END_IF

310: (* Warten auf Solldrehzahl erreicht *)

	IF (gpAx[nHliAxIfcIdx]^.lr_state.rev_erreicht_r) THEN
		nState := 0;
	END_IF


END_CASE


(*
IF nLogAxisNr <> 0 THEN
	IF pAC[nLogAxisNr] <> 0  THEN
		IF ADR(gpAx[nLogAxisNr]^) <> 0  THEN
			IF gpAx[nLogAxisNr]^.ipo_state.X_SpindleAxis = TRUE THEN

				(* command spindle revolution *)
				IF fbRTrigStart.Q THEN
					pCommand := ADR(gpAx[nLogAxisNr]^.ipo_mc_control.MCControlExtToIpo_ExtToIpo);
					IF (nSpeed > 0) THEN
						pCommand^.command_w.D_VbProg :=  DINT_TO_UDINT((nSpeed * 360 / 60) * 1000)  ;(*Programmierter Satzvorschub in u/min*)
  						pCommand^.command_w.W_DrehInfo := 1;(* rechtslauf *)
					ELSE
						pCommand^.command_w.D_VbProg :=  DINT_TO_UDINT((-nSpeed * 360 / 60) * 1000)  ;(*Programmierter Satzvorschub in u/min*)
						pCommand^.command_w.W_DrehInfo := 0;(* linkslauf*)
					END_IF
					pCommand^.command_w.D_GeoGmFkt := 0;(*G- und M- Fkt.-Bitleiste*)
					pCommand^.command_w.W_SatzTyp := HLI_NC_MOVE_ENDLOS;(*Einer der Werte: HLI_NC_MOVE_LIN, HLI_NC_MOVREF, HLI_NC_MOVE_ENDLOS, HLI_NC_SPINDEL_STOP*)
					pCommand^.command_semaphor_rw := TRUE;
				END_IF
				(* command spindle revolution *)
				IF fbRTrigStop.Q THEN
					pCommand := ADR(gpAx[nLogAxisNr]^.ipo_mc_control.MCControlExtToIpo_ExtToIpo);
					pCommand^.command_w.D_VbProg := 600000000;(*Programmierter Satzvorschub*)
					pCommand^.command_w.D_GeoGmFkt := 0;(*G- und M- Fkt.-Bitleiste*)

					pCommand^.command_w.W_SatzTyp := HLI_NC_SPINDEL_STOP;(*Einer der Werte: HLI_NC_MOVE_LIN, HLI_NC_MOVREF, HLI_NC_MOVE_ENDLOS, HLI_NC_SPINDEL_STOP*)
					pCommand^.command_w.W_DrehInfo := 0;(*Drehinformation*)
					pCommand^.command_semaphor_rw := TRUE;
				END_IF
			END_IF
		END_IF
	END_IF
END_IF
*)

END_FUNCTION_BLOCK

// ---- CNC Beckhoff/9 Mis/PB_10_CNC_Spindelkopplung.TcPOU
PROGRAM PB_10_CNC_Spindelkopplung
VAR
	pCoupling: POINTER TO HLI_COMMAND_AXIS_COUPLING;
	p_AxisCouplingState: POINTER TO HLI_STATE_AXIS_COUPLING;
	nState: INT;
	bBusy: BOOL;
	fbRTrig: R_TRIG;
	bCouple: BOOL;
	fbFTrig: F_TRIG;
END_VAR

(* allow axis coupling *)
gpAx[5]^.lr_mc_control.axis_coupling.enable_w := TRUE;


pCoupling := ADR(gpAx[5]^.lr_mc_control.axis_coupling.command_w);
p_AxisCouplingState := ADR(gpAx[5]^.lr_mc_control.axis_coupling.state_r);


fbRTrig(clk := bCouple);
fbFTrig(clk := bCouple);


IF (fbRTrig.Q) THEN			(* start coupling *)
	pCoupling^.desc[0].mode  := HLI_AXIS_COUPLING_DIRECT;
	pCoupling^.desc[0].ax_nr := 5;
	bBusy := TRUE;
	nState := 10;
END_IF


IF (fbFTrig.Q) THEN		(* end coupling *)
	pCoupling^.desc[0].mode  := HLI_AXIS_COUPLING_INACTIVE;
	pCoupling^.desc[0].ax_nr := 0;
	bBusy := TRUE;
	nState := 10; 
END_IF




CASE nState OF

0: (*IDLE *)
	bBusy := FALSE;


10: (* Koppeln oder Enkoppeln starten *)
	pCoupling^.semaphor_rw := TRUE;
	nState := nState + 10;

20:	(* Warten auf Koppeln fertig *)
	IF (pCoupling^.semaphor_rw = FALSE) THEN
		nState := 0;
	END_IF


END_CASE

END_PROGRAM

// ---- CNC Beckhoff/9 Mis/HLI3_ResetSpindle.TcPOU
FUNCTION HLI3_ResetSpindle : BOOL
VAR_INPUT
	/// axis number of spindle 
	nHliAxisIdx: INT;
END_VAR
VAR
	/// Index of axis specific HLI area 
	nHliAxIfcIdx: INT;
	SpdlState: BOOL;
	SpdlCommand: BOOL;
	ResetCmd: BOOL := FALSE;
	/// local pointer to data of actual axis 
	pResetUnit: POINTER TO MC_CONTROL_BOOL_UNIT;
END_VAR

HLI3_ResetSpindle := FALSE;

IF NOT HLI3_CheckAxisValid(nHliAxisIdx := nHliAxisIdx) THEN
	HLI3_ResetSpindle := FALSE;
	RETURN;
END_IF

	pResetUnit := ADR(gpAx[nHliAxisIdx]^.ipo_mc_control.spdl_reset);
	SpdlState  := pResetUnit^.state_r;

	IF ResetCmd = TRUE THEN
		pResetUnit^.command_w := TRUE;
		SpdlCommand           := pResetUnit^.command_w;
		HLI3_ResetSpindle          := SpdlState;
	END_IF

END_FUNCTION

// ---- CNC Beckhoff/Demo/PRG_Demo.TcPOU
PROGRAM PRG_Demo
VAR
	sLine1: STRING;
	sLine2: STRING;
	fbWriteZeroFddefault: FB_WriteCNCZeroOffsetDefault;
	bTest: BOOL;
	fbReadActiceG: HLI3_GetChannelActiveG;
	
	bReadG: BOOL;
	
END_VAR

PRG_MachineStatusV2();


sLine1 := 'Test line 1';
sLine2 := 'Test line two';

fbWriteZeroFddefault(
	bExecute:= bTest, 
	nG159Index:= 5 , 
	nChanIdx:=0, 
	bBusy=> , 
	bError=> , 
	nErrorID=> );
	
	
fbReadActiceG(
	bExec:= bReadG, 
	nChanIdx:= 0 , 
	ActiveG=> , 
	bBusy=> , 
	bError=> , 
	nErrorID=> );	
	
;

END_PROGRAM

// ---- CNC Beckhoff/Demo/PRG_MachineStatusV2.TcPOU
PROGRAM PRG_MachineStatusV2
VAR	
	fbTon: TON;
	fbTon2: TON;
	btest: BOOL;
	sName: STRING;
	sFarbe: STRING;
	nFarbe : UDINT;
	nFarbe2: UDINT;
	value: UDINT;
	value2 : UDINT;
	bUp: BOOL;
END_VAR


fbTon(in := NOT fbton.Q, pt := t#250ms);
IF (fbTon.Q) THEN
	btest := NOT bTest;
END_IF

fbton2(in := NOT fbton2.Q, pt := t#30ms);
IF fbton2.Q THEN

	IF (bUp) THEN
		value := value + 1;
	ELSE
		value := value - 1;
	END_IF
	IF value >= 200 THEN
		bUp := FALSE;
		value := 200;
	END_IF
	IF value <= 0 THEN
		bUp := TRUE;
		value := 0;
	END_IF
	value2 := 100 - value;
END_IF

nFarbe2 := 16#FF000000 + value2 * 2 * 16#010000 + value * 2 * 16#01;

IF btest THEN
	sName := 'EIN';
	sFarbe := 'blau';
	nFarbe := 16#FF0000FF;
ELSE
	sName := 'aus';
	sFarbe := 'rot';
	nFarbe := 16#FFFF0000;

END_IF

END_PROGRAM

// ---- CNC Beckhoff/Messages/FB_EventLog.TcPOU
FUNCTION_BLOCK FB_EventLog
VAR_INPUT
	bEvent: BOOL;
	bEventQuit: BOOL;
	bReset: BOOL;
	eLogMethod: E_LogMethod := Static;
	nSourceId: UDINT;
	nEventId: UDINT;
	nEventDataAddr: UDINT;
	nEventDataSize: UDINT;
	sFormat: STRING;
END_VAR
VAR_OUTPUT
	nEventState: UDINT;
	bEventActive: BOOL;
	bError: BOOL;
	nErrorId: UDINT;
END_VAR
VAR
	bEventInternal: BOOL;
	bEventActiveInternal: BOOL;
	fbFtrigEvent: F_TRIG;
	fbRtrigEvent: R_TRIG;
	fbRtrigEventInternal: R_TRIG;
	stEventData: TcEvent;
	fbEventLogger: ADSLOGEVENT;
END_VAR

(******************************************************************************)
(* 								 Konfiguration des Events									*)
(******************************************************************************)
stEventData.Flags 					:= TCEVENTFLAG_LOG OR TCEVENTFLAG_SRCID OR TCEVENTFLAG_FMTSELF OR 16#1000;
stEventData.StreamType				:= TCEVENTSTREAM_SIMPLE;
stEventData.ProgId 					:= 'TcEventFormatter.TcXmlFormatter';
stEventData.Id 						:= nEventId;
stEventData.SourceId 				:= nSourceId;
stEventData.DataFormatStrAddress	:= ADR(sFormat);
stEventData.bQuitRequired 			:= TRUE;

(******************************************************************************)
(* 					Interne Bildung des eventausloesenden Signals					*)
(******************************************************************************)
fbFtrigEvent
	(CLK := bEvent);

fbRtrigEvent
	(CLK := bEvent);

bEventInternal	:= (bEvent AND (eLogMethod = Static)) OR
					   (fbFtrigEvent.Q AND (eLogMethod = FallingTrig)) OR
					   (fbRtrigEvent.Q AND (eLogMethod = RisingTrig));

fbRtrigEventInternal
	(CLK := bEventInternal);

IF fbRtrigEventInternal.Q THEN
	bEventActiveInternal	:= TRUE;
ELSIF (fbEventLogger.EventState > 0) THEN
	bEventActiveInternal	:= FALSE;
END_IF

(******************************************************************************)
(* 							  Uebergabe an den Eventlogger								*)
(******************************************************************************)
fbEventLogger
	(NETID						:= '',
	 PORT						:= 110,
	 Event						:= bEventInternal,
	 EventQuit					:= bEventQuit,
	 EventConfigData			:= stEventData,
	 EventDataAddress			:= nEventDataAddr,
	 EventDataLength			:= nEventDataSize,
	 FbCleanup 					:= bReset,
	 TMOUT						:= t#2s,
	 EventState					=> nEventState,
	 Err						=> bError,
	 ErrId						=> nErrorId
	);

bEventActive					:= (fbEventLogger.EventState > 0) OR bEventActiveInternal;

END_FUNCTION_BLOCK

// ---- CNC Beckhoff/Messages/FB_ExtSimpleEventLog.TcPOU
///****************************************************************************************
///Name:				FB_ExtSimpleEventLog
///Date:				13.10.2004
///Author:			Dirk Nordberg (BECKHOFF INDUSTRIE ELEKTRONIK)
///
///Description: Function block to control the EventLogger
///	Messages can be activated or deactivated through an array of bool.
///	The subscription of the array is equivalent to EventID from EventLogger.
///	Funtion block will be initialized with Init flag, then the busy flag is set true. 
///
///	Revision:	1.3
///	History:		13.10.2004	Ng	start coding
///				17.04.2005	MK	runtime optimized
///				06.09.2005 	MiB extended version (renamed to FB_ExtSimpleEventLog)

///****************************************************************************************
FUNCTION_BLOCK FB_ExtSimpleEventLog
VAR_INPUT
	/// Rising flag starts the initialization 
	Init: BOOL;
	/// Alarm error class 
	Class: UINT;
	/// Activate or deaktivate confirmation 
	QuitRequired: BOOL;
	/// Adress of the array for the messages 
	adrAlarmArray: POINTER TO BOOL;
	/// ...with constant boundaries ARRAY_LBOUND to ARRAY_UBOUND for array size 
	adrQuitArray: POINTER TO BOOL;
	/// ...with constant boundaries ARRAY_LBOUND to ARRAY_UBOUND for array size 
	adrEventData: POINTER TO ST_EventData;
END_VAR
VAR_OUTPUT
	Busy: BOOL;
	Err: BOOL;
	ErrId: UDINT;
END_VAR
VAR CONSTANT
	ARRAY_LBOUND: UDINT := FIRST_MESSAGE;
	ARRAY_UBOUND: UDINT := LAST_MESSAGE;
	TCEVENTDATAFORMATSTRING: STRING(80) := ' ';
	STATE_INIT: INT := 0;
	STATE_IDLE: INT := 1;
	STATE_RESET_EVENT: INT := 2;
	STATE_QUIT_EVENT: INT := 3;
	STATE_RESET_END: INT := 4;
	STATE_WAIT: INT := 5;
END_VAR
VAR
	state: INT;
	///{flag nowatch on }
	bReady: BOOL;
	nMsgHasChanged: DINT;
	bEvtState: ARRAY[ARRAY_LBOUND..ARRAY_UBOUND] OF BOOL;
	event: ARRAY[ARRAY_LBOUND..ARRAY_UBOUND] OF ADSLOGEVENT;
	idx: UDINT;
	CfgEvent: TcEvent;
	bWait: BOOL;
	ptAlarm: POINTER TO BOOL;
	ptQuit: POINTER TO BOOL;
	RT_Init: R_TRIG;
	ptData: POINTER TO ST_EventData;
	stDummy: ST_EventData;
	/// Format String for message 
	sFormatString: STRING := '';
	arrParaPointer: ARRAY[1..5] OF POINTER TO UDINT;
	nPara1: DINT;
	sPara2: STRING;
	sPara3: STRING;
	sPara4: STRING;
	sPara5: STRING;
END_VAR

nMsgHasChanged := MEMCMP(ADR(bEvtState), adrAlarmArray, SIZEOF(bEvtState));
RT_Init(CLK:=Init);

CASE State OF
	STATE_INIT:		(* Set the parameter for TcEvent *)
		Err := FALSE;
		ErrId :=0;
		Busy := FALSE;
		CfgEvent.Prio := 0;
		CfgEvent.DataFormatStrAddress := ADR(TCEVENTDATAFORMATSTRING);
		CfgEvent.Flags := TCEVENTFLAG_LOG OR TCEVENTFLAG_SRCID;
		CfgEvent.StreamType := TCEVENTSTREAM_SIMPLE;
		CfgEvent.ProgId := 'TcEventFormatter.TcXmlFormatter';
		CfgEvent.SourceId := nSourcePlc;
	(*	CfgEvent.Class := Class ; *)
		CfgEvent.bQuitRequired := QuitRequired;
		FOR idx := ARRAY_LBOUND TO ARRAY_UBOUND BY 1 DO
			CfgEvent.Id := idx;
			event[idx](NETID:='', PORT:=110, Event:=FALSE , EventQuit:=FALSE,
				 EventConfigData:=CfgEvent, FbCleanup:=FALSE, TMOUT:=t#1s);
		END_FOR;
		State := STATE_IDLE;

	STATE_IDLE:
		(* nothing to do *)
		IF nMsgHasChanged = 0 AND NOT RT_Init.Q THEN
			RETURN;
		END_IF

		IF adrAlarmArray <> 0 THEN
			ptAlarm := adrAlarmArray;
			ptData := adrEventData;
			IF ptData <> 0 THEN
				sFormatString := '%d%s%s%s%s';
				FOR idx := ARRAY_LBOUND TO ARRAY_UBOUND BY 1 DO

					nPara1 := UDINT_TO_DINT(ptData^.nErrorCode);
	
					sPara2 := CONCAT('[S',UINT_TO_STRING(ptData^.nSourceText));
					sPara2 := CONCAT(sPara2,'E');
					sPara2 := CONCAT(sPara2,UDINT_TO_STRING(ptData^.nErrorCode));
					sPara2 := CONCAT(sPara2,']');
	
			  		sPara3 := CONCAT('[S',UINT_TO_STRING(ptData^.nSourceDesc));
					sPara3 := CONCAT(sPara3,'E');
					sPara3 := CONCAT(sPara3,UDINT_TO_STRING(ptData^.nErrorCode));
					sPara3 := CONCAT(sPara3,']');
	
					sPara4 := ptData^.sModul;
					sPara5 := ptData^.sAddInfo;
	
					arrParaPointer[1] := ADR(nPara1);
					arrParaPointer[2] := ADR(sPara2);
					arrParaPointer[3] := ADR(sPara3);
					arrParaPointer[4] := ADR(sPara4);
					arrParaPointer[5] := ADR(sPara5);
	
					event[idx].EventConfigData.DataFormatStrAddress := ADR(sFormatString);
					event[idx].EventConfigData.Id := nEventPlc;
					event[idx].EventConfigData.SourceId := nSourcePlc ;
					event[idx].EventDataAddress := ADR(arrParaPointer);
					event[idx].EventDataLength := 0;

					event[idx]();
					ptData := ptData + SIZEOF(stDummy);
				END_FOR
			END_IF
			IF CfgEvent.bQuitRequired AND adrQuitArray <> 0 THEN
				ptQuit := adrQuitArray;
				FOR idx := ARRAY_LBOUND TO ARRAY_UBOUND BY 1 DO
					event[idx](Event:=ptAlarm^, EventQuit:=ptQuit^);
					ptAlarm := ptAlarm + 1;
					ptQuit := ptQuit + 1;
				END_FOR;
			ELSE
				bReady := TRUE;
				FOR idx := ARRAY_LBOUND TO ARRAY_UBOUND BY 1 DO
					event[idx](Event:=ptAlarm^);
					ptAlarm := ptAlarm + 1;
					IF (NOT(event[idx].Event = TRUE			(* event is set *)
							AND event[idx].Quit = FALSE
							AND event[idx].EventState = TCEVENTSTATE_SIGNALED)
						AND NOT(event[idx].Event = FALSE		(* event is reset *)
							AND event[idx].Quit = TRUE
							AND event[idx].EventState = TCEVENTSTATE_INVALID)) THEN
						bReady := FALSE;
					END_IF
				END_FOR;

				(* copy the status *)
				IF bReady THEN
					MEMCPY(ADR(bEvtState), adrAlarmArray, SIZEOF(bEvtState));
				END_IF

			END_IF
		END_IF

		IF RT_Init.Q THEN
			Busy := TRUE;
			State := STATE_RESET_EVENT;
		END_IF

	STATE_RESET_EVENT:(*---------------------------------- clear messages ----------------------------------------*)
		FOR idx := ARRAY_LBOUND TO ARRAY_UBOUND BY 1 DO
			IF event[idx].EventState = TCEVENTSTATE_SIGNALED THEN
				event[idx](Event:=FALSE, EventQuit:= FALSE, FbCleanup:= FALSE, TMOUT:= t#1s);
				IF event[idx].Err THEN
					Err := TRUE;
					ErrId := event[idx].ErrId;
					IF event[idx].ErrId = 1282 THEN	(* Message Router: mailbox full *)
						event[idx](Event:=FALSE, EventQuit:= FALSE, FbCleanup:= FALSE);
						RETURN;
					END_IF
				END_IF
			END_IF;
		END_FOR;
		State := STATE_QUIT_EVENT;

	STATE_QUIT_EVENT:(*---------------------------------- quit messages ----------------------------------------*)
		FOR idx := ARRAY_LBOUND TO ARRAY_UBOUND BY 1 DO
			IF event[idx].EventState = TCEVENTSTATE_SIGNALED THEN
				event[idx](Event:=FALSE, EventQuit:= TRUE, FbCleanup:= FALSE, TMOUT:= t#1s);
				IF event[idx].Err THEN
					Err := TRUE;
					ErrId := event[idx].ErrId;
					IF event[idx].ErrId = 1282 THEN	(* Message Router: mailbox full *)
						event[idx](Event:=FALSE, EventQuit:= FALSE, FbCleanup:= FALSE);
						RETURN;
					END_IF
				END_IF
			END_IF;
		END_FOR;
		State := STATE_RESET_END;

	STATE_RESET_END:
		bWait := FALSE;
		FOR idx := ARRAY_LBOUND TO ARRAY_UBOUND BY 1 DO
			event[idx](Event:=FALSE, EventQuit:= FALSE, FbCleanup:= FALSE);
			IF event[idx].EventState = TCEVENTSTATE_SIGNALED THEN
				bWait := TRUE;
			END_IF
		END_FOR;
		IF NOT bWait THEN
			State := STATE_INIT;
		END_IF

END_CASE

END_FUNCTION_BLOCK

// ---- CNC Beckhoff/Util/Blinker.TcPOU
FUNCTION_BLOCK Blinker
VAR_INPUT
	Taktzeit: TIME;
END_VAR
VAR_OUTPUT
	Ausgang: BOOL;
END_VAR
VAR
	Timer1: TON;
END_VAR

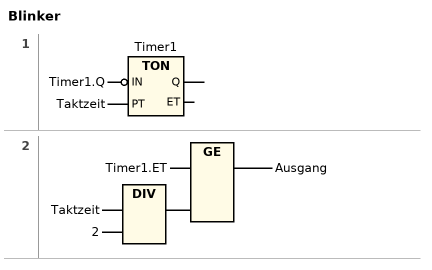
// NETWORK 1
Timer1(IN := NOT Timer1.Q, PT := Taktzeit); // TON

// NETWORK 2
Ausgang := Timer1.ET >= Taktzeit / 2;

END_FUNCTION_BLOCK

// ---- CNC Beckhoff/Util/FB_CNCWriteParameter.TcPOU
///*********************************************************************************************************
///NAME.......................:		FB_CNCWriteParameter
///DATUM....................:			03.07.2015
///AUTOR....................:			Thomas Voß
///VERSION................:			1.2
///
///Description.: 	The function block allows to write cnc parameters to the CNC kernel.					
///**********************************************************************************************************
FUNCTION_BLOCK FB_CNCWriteParameter
VAR_INPUT
	/// Channel Id
	nChannelId: UINT;
	/// log. Axis Id  
	nLogAxisId: UINT;
	bExecute: BOOL;
	/// numbers of parameters 
	nNumParameters: INT;
	/// Parameter type
	eParameterType: E_CNCParameterTypes;
	/// Windows temp file for sub lists
	strTempPath: STRING;
END_VAR
VAR_OUTPUT
	bBusy: BOOL;
	bError: BOOL;
	nErrorID: INT;
END_VAR
VAR_IN_OUT
	stParameter: ARRAY[1..200] OF ST_CNCParameter;
END_VAR
VAR
	fbOnTrigger: R_TRIG;
	Step: UDINT;
	FbAdsWrite: ADSWRITE;
	strParameterLine: STRING(255);
	strFileName: STRING(255);
	strHeader: STRING(255);
	TimeOut: TON;
	m: DINT;
	/// Text To File 
	fbFileOpen: FB_FileOpen;
	fbFileRead: FB_FileRead;
	fbFilePuts: FB_FilePuts;
	fbFileClose: FB_FileClose;
	hFileOutput: UINT := 0;
END_VAR
VAR CONSTANT
	nMaxParameters: INT := 200;
	/// Ads Interface 
	nAdsPortNumber: UINT := 553;
	nAdsIndexGroup: UDINT := 16#20100;
	nAdsIndexGroupAxisParameter: UDINT := 16#20200;
	nAdsIndexOffsetlogAxisNumber: UDINT := 16#37;
	nAdsIndexOffsetChannelParameter: UDINT := 16#34;	
	nAdsIndexOffsetAxisParameter: UDINT := 16#18;
	nAdsIndexOffsetZeroOffsets: UDINT := 16#2E;
	nAdsIndexOffsetToolParameter: UDINT := 16#30;
	nAdsIndexOffsetClampPosition: UDINT := 16#32;
	nAdsIndexOffsetCompensationTable: UDINT := 16#39;
	/// Time Out Error 
	ErrID_1: INT := 1;
	/// Fehler beim Öffnen der Parameterdatei 
	ErrID_2: INT := 2;
	/// ADS - Fehler : Vorgabe Achs ID 
	ErrID_3: INT := 3;
	/// ADS - Fehler : Aktivierung der Parameterliste 
	ErrID_4: INT := 4;
	/// Invalid   CNC Parameter Type 
	ErrID_5: INT := 5;
	/// Invalid   Axis Number  
	ErrID_6: INT := 6;
	/// Invalid   Channel Number  
	ErrID_7: INT := 7;
	/// Invalid   Number  of Parameters 
	ErrID_8: INT := 8;
	/// File Error 
	ErrID_9: INT := 9;
	/// Invalid Channel State 
	ErrID_10: INT := 10;
END_VAR



fbOnTrigger(CLK:= bExecute);

IF fbOnTrigger.Q THEN
	Step 	:= 10;
	nErrorID 	:= 0;
	bError	 := 0;
	bBusy := TRUE;
END_IF

CASE Step OF
0:
	bBusy := FALSE;

10: (* check input parameters *)
	IF (nNumParameters < 1 OR nNumParameters > nMaxParameters) THEN
		nErrorID 	:= ErrID_8;
		Step := 999;
	ELSE
		CASE eParameterType OF
				
			CNC_AxisParameter:
				IF (nLogAxisId <= 0  OR nLogAxisId > 64) THEN
					nErrorID 	:= ErrID_6;
					Step := 999;
	
				ELSIF (nChannelID <= 0 OR nChannelID	 > 12	) THEN
					nErrorID 	:= ErrID_7;
					Step := 999;
				ELSE
					Step := 12;
				END_IF

			CNC_ChannelParameter:
				IF (nChannelID <= 0 OR nChannelID > 12) THEN
					nErrorID 	:= ErrID_7;
					Step := 999;
				ELSE
					Step := 12;
				END_IF

			CNC_ToolParameter:
				IF (nChannelID <= 0 OR nChannelID > 12) THEN
					nErrorID 	:= ErrID_7;
					Step := 999;
				ELSE
					Step := 12;
				END_IF
	
			CNC_ClampPosition:
				IF (nChannelID <= 0 OR nChannelID > 12) THEN
					nErrorID 	:= ErrID_7;
					Step := 999;
				ELSE
					Step := 12;
				END_IF
	
			CNC_ZeroOffsets:
				IF (nChannelID <= 0 OR nChannelID > 12) THEN
					nErrorID 	:= ErrID_7;
					Step := 999;
				ELSE
					Step := 12;
				END_IF
		END_CASE
	END_IF

	fbFileOpen.bExecute := FALSE;
	
	// Check Channel State
	IF (cncSystem.Channel[nChannelId-1].ActState <> HLI_IMCM_PROCESS_SELECTED AND 
		cncSystem.Channel[nChannelId-1].ActState <> HLI_IMCM_PROCESS_READY) THEN
		nErrorID 	:= ErrID_10;
		Step := 999;
	END_IF

12:	(* create file name and list file header  *)
	strHeader := '';

	CASE eParameterType OF

		CNC_AxisParameter:
			strFileName := CONCAT(strTempPath, '\axis');
			strFileName := CONCAT(strFileName, UINT_TO_STRING(nLogAxisId));
			strFileName := CONCAT(strFileName, '.lis');

			strHeader := 'kopf.achs_nr ';
			strHeader := CONCAT(strHeader, UINT_TO_STRING(nLogAxisId));
			Step := 15;
		CNC_ChannelParameter:
			strFileName := CONCAT(strTempPath, '\channel');			
			strFileName := CONCAT(strFileName, UINT_TO_STRING(nChannelID));
			strFileName := CONCAT(strFileName, '.lis');
			Step := 15;
		CNC_ToolParameter:			
			strFileName := CONCAT(strTempPath, '\ToolCh');
			strFileName := CONCAT(strFileName, UINT_TO_STRING(nChannelID));
			strFileName := CONCAT(strFileName, '.lis');
			Step := 15;
		CNC_ClampPosition:
			strFileName := CONCAT(strTempPath, '\ClampPosCh');			
			strFileName := CONCAT(strFileName, UINT_TO_STRING(nChannelID));
			strFileName := CONCAT(strFileName, '.lis');
			Step := 15;
		CNC_ZeroOffsets:			
			strFileName := CONCAT(strTempPath, '\ZeroOffsetsChh');
			strFileName := CONCAT(strFileName, UINT_TO_STRING(nChannelID));
			strFileName := CONCAT(strFileName, '.lis');
			Step := 15;
		ELSE
			nErrorID 	:= ErrID_5;
			Step := 999;
	END_CASE

15:	(* write file to destination folder *)
	fbFileOpen.sNetId := '';
	fbFileOpen.sPathName := strFileName;
	fbFileOpen.nMode := FOPEN_MODEWRITE OR FOPEN_MODETEXT;
	fbFileOpen.ePath := PATH_GENERIC;
	fbFileOpen.tTimeout := t#1s;
	fbFileOpen.bExecute := TRUE;
	Step := 16;

16:
	IF ( NOT fbFileOpen.bBusy ) THEN
		IF ( fbFileOpen.bError ) THEN
			nErrorID  :=ErrID_9 ;
			bError := TRUE;
			Step := 999;
		ELSE
			hFileOutput := fbFileOpen.hFile;
			fbFilePuts.bExecute:= FALSE;
			Step := 17;
		END_IF
	END_IF


17: (* Write Header File *)
	fbFilePuts.sNetId:='';
	fbFilePuts.hFile:=hFileOutput;
	fbFilePuts.bExecute:=TRUE;
	fbFilePuts.tTimeout:=t#10s;
	fbFilePuts.sLine :=strHeader;
	Step := 18;

18:
	IF ( NOT fbFilePuts.bBusy ) THEN
		IF ( fbFilePuts.bError ) THEN
			 nErrorID  :=ErrID_9 ;
			bError := TRUE;
			Step := 999;
		ELSE
			fbFilePuts.bExecute:= FALSE;
			m := 1;
			Step := 19;
		END_IF
	END_IF


19:	(* Write Parameter lines *)
		strParameterLine :=  CONCAT('$N',stParameter[m].strName);
		strParameterLine :=  CONCAT(strParameterLine,'   ');
		strParameterLine := CONCAT(strParameterLine, stParameter[m].strValue);
		fbFilePuts.sLine :=strParameterLine;
		fbFilePuts.bExecute:= TRUE;
		Step := 20;
20:
		IF ( NOT fbFilePuts.bBusy ) THEN
			IF ( fbFilePuts.bError ) THEN
				 nErrorID  :=ErrID_9 ;
				bError := TRUE;
				Step := 999;
			ELSE
				Step := 21;
			END_IF
		END_IF

21:	(* Next Line *)
	IF (m+1 <= nMaxParameters AND m+1 <= nNumParameters) THEN
		m := m+1;
		fbFilePuts.bExecute:= FALSE;
		Step := 19;
	ELSE
		fbFilePuts.bExecute:= FALSE;
		Step := 22;
	END_IF

22:	(* Write footer *)
	fbFilePuts.sLine :='$NEnde';
	fbFilePuts.bExecute:= TRUE;
	Step := 23;

23:
	IF ( NOT fbFilePuts.bBusy ) THEN
		IF ( fbFilePuts.bError ) THEN
			 nErrorID  :=ErrID_9 ;
			bError := TRUE;
			Step := 999;
		ELSE
			fbFileClose.bExecute:=FALSE;
			Step := 30;
		END_IF
	END_IF


30:	(* Close File *)
	fbFileClose.sNetId:='';
	fbFileClose.hFile:=hFileOutput;
	fbFileClose.bExecute:=TRUE;
	fbFileClose.tTimeout:=t#1s;

	IF ( NOT fbFileClose.bBusy ) THEN
		IF ( fbFileClose.bError ) THEN
			 nErrorID  :=ErrID_9 ;
			bError := TRUE;
			Step := 999;
		ELSE
			hFileOutput := 0;
			Step := 35;
		END_IF
	END_IF

	35:
		CASE eParameterType OF
			CNC_AxisParameter:
				Step := 60;
			CNC_ChannelParameter:
				Step := 60;
			CNC_ToolParameter:
				Step := 60;
			CNC_ClampPosition:
				Step := 60;
			CNC_ZeroOffsets:
				Step := 60;
		END_CASE

	40:	(* logical axis ID*)
		TimeOut(IN:=FALSE);
		FbAdsWrite( Port := 553, IdxGrp := nAdsIndexGroup  + nChannelID, IdxOffs := (nAdsIndexOffsetlogAxisNumber), LEN := SIZEOF(nLogAxisID), SrcAddr := ADR(nLogAxisID),TMOUT := T#1S, WRITE := TRUE);
		Step := 50;
	50:
		TimeOut(IN:=TRUE, PT:=T#2S);

		FbAdsWrite();
		IF FbAdsWrite.BUSY = FALSE THEN
			IF NOT FbAdsWrite.ERR THEN
				FbAdsWrite( WRITE := FALSE);
				Step := 60;
			ELSE
				FbAdsWrite( WRITE := FALSE);
				nErrorID := ErrID_3;
				Step := 999;
			END_IF
		END_IF

		(* error timeout *)
		IF TimeOut.Q THEN
			nErrorID 	:= ErrID_1;
			Step   	:= 999;
		END_IF

	60:	(* activate List File *)
		TimeOut(IN:=FALSE);

		CASE eParameterType OF

		CNC_AxisParameter:
			FbAdsWrite( Port := nAdsPortNumber, IdxGrp := nAdsIndexGroupAxisParameter  + nLogAxisId, IdxOffs := (nAdsIndexOffsetAxisParameter), LEN := SIZEOF(strFileName), SrcAddr := ADR(strFileName), WRITE := TRUE);
		CNC_ChannelParameter:
			FbAdsWrite( Port := nAdsPortNumber, IdxGrp := nAdsIndexGroup  + nChannelID, IdxOffs := (nAdsIndexOffsetChannelParameter), LEN := SIZEOF(strFileName), SrcAddr := ADR(strFileName), WRITE := TRUE);
		CNC_ToolParameter:
			FbAdsWrite( Port := nAdsPortNumber, IdxGrp := nAdsIndexGroup  + nChannelID, IdxOffs := (nAdsIndexOffsetToolParameter), LEN := SIZEOF(strFileName), SrcAddr := ADR(strFileName), WRITE := TRUE);
		CNC_ClampPosition:
			FbAdsWrite( Port := nAdsPortNumber, IdxGrp := nAdsIndexGroup  + nChannelID, IdxOffs := (nAdsIndexOffsetClampPosition), LEN := SIZEOF(strFileName), SrcAddr := ADR(strFileName), WRITE := TRUE);
		CNC_ZeroOffsets:
			FbAdsWrite( Port := nAdsPortNumber, IdxGrp := nAdsIndexGroup  + nChannelID, IdxOffs := (nAdsIndexOffsetZeroOffsets), LEN := SIZEOF(strFileName), SrcAddr := ADR(strFileName), WRITE := TRUE);
		END_CASE

		Step := 70;
	70:
		TimeOut(IN:=TRUE, PT:=T#2S);
		FbAdsWrite();
		IF FbAdsWrite.BUSY = FALSE THEN

			IF NOT FbAdsWrite.ERR THEN
				FbAdsWrite( WRITE := FALSE);
				Step := 0;
			ELSE
				FbAdsWrite( WRITE := FALSE);
				nErrorID := ErrID_4;
				Step := 999;
			END_IF
		END_IF

		(* error timeout *)
		IF TimeOut.Q THEN
			nErrorID 	:= ErrID_1;
			Step   	:= 999;
		END_IF

999: (* Fehler *)
		bBusy  := FALSE;
		bError := TRUE;
		Step 	 := 0;
END_CASE

fbFileOpen();
fbFilePuts();
fbFileClose();

END_FUNCTION_BLOCK

// ---- CNC Beckhoff/Util/F_GRAYCODE_TO_UINT.TcPOU
FUNCTION F_GRAYCODE_TO_UINT : UINT
VAR_INPUT
	byGraycodeSwitches	: BYTE;
END_VAR
VAR
	nLoopCount				: INT;
	byResult					: BYTE;
	bySwitches				: BYTE;
END_VAR

bySwitches			:= byGraycodeSwitches;
byResult				:= 0;

FOR nLoopCount := 0 TO 31 DO
	byResult 		:= byResult XOR bySwitches;
	bySwitches		:= SHR(bySwitches, 1);
END_FOR

F_GRAYCODE_TO_UINT	:= BYTE_TO_UINT(byResult);

END_FUNCTION

// ---- CNC Beckhoff/Util/HLI3_FindHliAxisIdx.TcPOU
FUNCTION HLI3_FindHliAxisIdx : DINT
VAR_INPUT
	nLogAxisNo		: UDINT;	
END_VAR
VAR
	i				: UINT;	
END_VAR

IF nLogAxisNo > MAX_SYS_LOG_AXIS_INDEX OR nLogAxisNo < 1 THEN 
	HLI3_FindHliAxisIdx := -1;
ELSE
	HLI3_FindHliAxisIdx := CNCSystem.LogAxisNo[nLogAxisNo].nHliAxisIdx;	
END_IF

END_FUNCTION

// ---- CNC Beckhoff/Util/HLI3_FindAxisNameAndChannel.TcPOU
FUNCTION HLI3_FindAxisNameAndChannel : BOOL
VAR_INPUT
	LogAxeNr		: UDINT;
	pAxisName		: POINTER TO STRING(HLI_ACHS_NAME_LAENGE);
	pChannelNr		: POINTER TO UINT;
END_VAR
VAR
	i				: UDINT;
	
	pString			: POINTER TO STRING;
END_VAR

FOR i := 0 TO gNrAx - 1 DO
	IF gpAx[i]^.ipo_state.log_achs_nr_r = LogAxeNr THEN
		pChannelNr^ := gpAx[i]^.ipo_state.cnc_channel_r;	(* channel of axis *)
		FOR i := 0 TO INT_TO_UDINT(HLI_CH_AX_MAXIDX) DO
			IF gpCh[pChannelNr^-1]^.bahn_state.coord_r[i].log_achs_nr_r = LogAxeNr THEN
				pString                := ADR(gpCh[pChannelNr^-1]^.bahn_state.coord_r[i].axis_name_r.zeichen);	(* name of axis *)
				pAxisName^             := pString^;
				HLI3_FindAxisNameAndChannel := TRUE;
				RETURN;
			END_IF
		END_FOR
	END_IF
END_FOR

pAxisName^ := '';
pChannelNr^ := 0;
HLI3_FindAxisNameAndChannel := FALSE;

END_FUNCTION
